Yaskawa INFORM job: OK_R2_O242(-90,180)OKKR.JBI

/JOB
//NAME OK_R2_O242(-90,180)OKKR
///FOLDERNAME X4
//POS
///NPOS 132,132,132,4,0,0
///TOOL 0
///POSTYPE PULSE
///PULSE
C00000=-1085,-105763,-105592,-1367,57789,79187
C00001=-48587,-61870,-56373,-37554,57186,71211
C00002=-109319,-98863,-81663,17130,36799,47258
C00003=-110499,-70978,-76585,14581,28064,55521
C00004=-114923,11399,-23396,32739,57115,42289
C00005=-116623,27529,-9023,35345,61036,36673
C00006=-106531,29443,-6029,23966,54360,54184
C00007=-107072,29107,-4870,24608,53702,53789
C00008=-107072,28853,-4001,24811,53095,53633
C00009=-107072,28916,-4224,24758,53250,53673
C00010=-107722,30543,-2610,25264,53294,53401
C00011=-107072,28916,-4224,24758,53250,53673
C00012=-111142,26244,-323,41203,47920,52388
C00013=-110370,28048,1439,40770,47447,52585
C00014=-111142,26244,-323,41203,47920,52388
C00015=-118906,20077,-8538,45056,52999,50729
C00016=-119909,26329,-1133,46362,52540,49898
C00017=-119909,26168,171,46853,51920,49532
C00018=-119909,26196,-79,46760,52037,49603
C00019=-119136,27214,914,46366,51584,49791
C00020=-119909,26334,-1167,46350,52555,49909
C00021=-114397,22245,-5862,42574,50447,51878
C00022=-114678,22860,-3308,43462,49647,51288
C00023=-115167,24031,-2185,43822,49818,51101
C00024=-114397,22245,-5862,42574,50447,51878
C00025=-121530,27687,-2626,46433,54487,50098
C00026=-123087,41300,13747,48930,53168,48397
C00027=-123087,41268,14126,49069,53001,48291
C00028=-123087,41187,15376,49530,52460,47945
C00029=-123087,41201,15124,49437,52567,48015
C00030=-122538,42735,16737,49268,52140,48077
C00031=-123087,41401,12757,48563,53611,48677
C00032=-122129,71626,35140,38253,65229,58469
C00033=-121790,71611,37598,38532,63876,58094
C00034=-121434,69636,35263,38247,64057,58328
C00035=-122129,71626,35140,38253,65229,58469
C00036=-120911,36076,-5205,37468,69020,59397
C00037=-115840,28901,-5746,41502,62039,42211
C00038=-98326,48101,7238,8655,64893,45952
C00039=-115260,32848,2305,42264,59563,41364
C00040=-114901,35009,3238,41874,59801,41652
C00041=-97533,41248,-17,1386,65111,50229
C00042=-97538,41207,-61,1389,65116,50227
C00043=-106518,42771,1588,20090,69082,39147
C00044=-114870,56219,16256,34532,77057,29376
C00045=-115508,58548,18881,34817,76955,29091
C00046=-119108,76539,39651,36547,75490,27151
C00047=-119068,69741,30113,36226,77407,27817
C00048=-119017,62946,18494,35839,80377,88071
C00049=-119017,62946,18494,34539,69439,88067
C00050=-120365,66463,30779,36511,65240,86054
C00051=-120262,68091,33866,36748,64342,85770
C00052=-120262,68091,33866,36748,64342,85770
C00053=-120199,73821,40919,37119,63187,85370
C00054=-119797,77336,44812,37019,63133,85550
C00055=-121282,70665,32992,36655,66863,86263
C00056=-119068,69741,30113,36226,77407,27817
C00057=-122206,59988,23685,43496,73319,20353
C00058=-127814,79238,36559,32495,95149,850
C00059=-120292,64376,19422,33176,77212,56642
C00060=-112530,30789,-557,20785,48585,51256
C00061=-109411,60829,14687,9556,77735,26746
C00062=-109666,62467,17842,9701,76678,26580
C00063=-109739,35424,4016,18642,47529,52303
C00064=-109346,36012,4533,18322,47429,52463
C00065=-111432,39361,576,18526,58483,53933
C00066=-120982,47505,9487,38936,66696,53604
C00067=-124164,44416,17003,51861,57678,49293
C00068=-125991,53710,27094,53356,57812,48240
C00069=-126351,53462,26814,53496,58041,48175
C00070=-128648,70270,46080,56033,57461,46239
C00071=-128914,63950,33868,51063,60408,47630
C00072=-125493,46290,11213,43702,62626,49802
C00073=-121024,34692,-8870,25769,64212,48636
C00074=-116968,-20453,-45092,25851,41430,48067
C00075=-118489,-78623,-76964,34127,32976,43558
C00076=-15896,-74508,-72271,-73191,84674,57421
C00077=-31461,-74136,-72097,-73237,111249,57325
C00078=-37199,-69408,-69826,-73614,107600,56062
C00079=3643,-76224,-106676,19950,71810,76872
C00080=-49550,-101636,-102264,-56737,88786,-31332
C00081=-138514,-74114,-82544,-4040,38797,-48213
C00082=-129498,7065,-37023,-9065,67369,-37181
C00083=-133542,65003,16374,-22570,90358,-433
C00084=-140622,86165,36573,-15496,97977,30873
C00085=-140802,90119,43938,-15362,95529,31124
C00086=-140802,89712,44636,-15338,94910,31202
C00087=-140802,89824,44435,-15345,95084,31180
C00088=-141302,92318,47595,-15241,94356,31104
C00089=-140802,90328,43607,-15371,95825,31086
C00090=-139449,100407,57298,-15497,92942,31904
C00091=-140520,104512,63149,-15296,91307,31746
C00092=-140782,103254,61503,-15262,91612,31621
C00093=-140520,104512,63149,-15296,91307,31746
C00094=-139554,101999,57136,-15503,93810,31760
C00095=-146528,71128,18474,-14629,100276,28663
C00096=-157576,61757,12077,-2365,89224,8186
C00097=-158570,72432,22020,-167,94145,8287
C00098=-158570,72037,22464,-167,93669,8287
C00099=-158570,72148,22336,-167,93805,8287
C00100=-157930,73423,23870,-319,93520,8487
C00101=-158570,72260,22211,-167,93940,8288
C00102=-159049,73117,23241,-53,93746,8137
C00103=-159487,76071,26810,51,93068,8000
C00104=-159049,73117,23241,-53,93746,8137
C00105=-152305,60889,6833,-1672,97624,10189
C00106=-140378,92804,43752,-12660,95661,26275
C00107=-136628,131083,97606,-23032,87536,68506
C00108=-138246,133972,103985,-22893,84834,68434
C00109=-138116,121410,87047,-22215,87119,66148
C00110=-138089,120831,86265,-22218,87298,66125
C00111=-139222,110925,72109,-17859,93005,38128
C00112=-141573,89787,44718,-13729,93335,28318
C00113=-147118,72338,23336,-11669,95813,24471
C00114=-147124,72286,23273,-11668,95824,24468
C00115=-156033,62541,11743,1459,94557,7242
C00116=-162183,69089,19251,9179,95274,-2750
C00117=-162693,76607,28216,6950,92750,113
C00118=-162306,74109,24034,6874,94001,304
C00119=-159278,70446,19892,6162,94440,1277
C00120=-158882,69844,19507,6067,94341,1397
C00121=-162546,67834,20044,10120,87741,415
C00122=-153853,64460,11220,-3191,96050,12949
C00123=-153394,69903,19674,-3303,93668,13156
C00124=-150617,75820,26688,-3977,92508,14059
C00125=-150141,75566,26453,-4094,92547,14205
C00126=-143887,90860,45319,-9758,90806,22100
C00127=-142426,78831,26541,-11541,97051,24087
C00128=-145972,26725,-27800,-4713,87219,24751
C00129=-154694,-16289,-62866,3052,73548,23707
C00130=-178421,-116488,-119781,18026,60210,14368
C00131=-104141,-125863,-97896,-54468,42310,-61417
BC00000=193639,675452,895426
BC00001=148805,682642,173588
BC00002=141606,703754,90547
BC00003=133760,726761,53
BC00004=133760,726761,53
BC00005=133760,726761,53
BC00006=133760,726761,53
BC00007=133760,726761,53
BC00008=133760,726761,53
BC00009=133760,726761,53
BC00010=133760,726761,53
BC00011=133760,726761,53
BC00012=133760,726761,53
BC00013=133760,726761,53
BC00014=133760,726761,53
BC00015=133760,726761,53
BC00016=133760,726761,53
BC00017=133760,726761,53
BC00018=133760,726761,53
BC00019=133760,726761,53
BC00020=133760,726761,53
BC00021=133760,726761,53
BC00022=133760,726761,53
BC00023=133760,726761,53
BC00024=133760,726761,53
BC00025=133760,726761,53
BC00026=133760,726761,53
BC00027=133760,726761,53
BC00028=133760,726761,53
BC00029=133760,726761,53
BC00030=133760,726761,53
BC00031=133760,726761,53
BC00032=133760,726761,53
BC00033=133760,726761,53
BC00034=133760,726761,53
BC00035=133760,726761,53
BC00036=133760,726761,53
BC00037=122204,725818,53
BC00038=122204,725818,53
BC00039=122204,725818,53
BC00040=122204,725818,53
BC00041=122204,725818,53
BC00042=122204,725818,53
BC00043=122204,725818,53
BC00044=122204,725818,53
BC00045=122204,725818,53
BC00046=122204,725818,53
BC00047=122204,725818,53
BC00048=122204,725818,53
BC00049=122204,725818,53
BC00050=122204,725818,53
BC00051=122204,725818,50
BC00052=122204,725818,50
BC00053=122204,725818,50
BC00054=122204,725818,50
BC00055=122204,725818,50
BC00056=122204,725818,53
BC00057=122204,725818,53
BC00058=171344,723534,1465
BC00059=151059,717900,51
BC00060=151059,717900,51
BC00061=151058,717899,53
BC00062=151058,717899,53
BC00063=151059,717900,51
BC00064=151059,717900,51
BC00065=151059,717900,51
BC00066=151059,717900,51
BC00067=151059,717900,51
BC00068=151059,717899,51
BC00069=151059,717900,51
BC00070=151059,717900,51
BC00071=151059,717900,51
BC00072=151059,717900,51
BC00073=150319,720693,10790
BC00074=145099,682085,7405
BC00075=145099,683773,7405
BC00076=139754,687631,3940
BC00077=139754,686805,3940
BC00078=139920,676862,3936
BC00079=199464,674570,1075173
BC00080=228966,680708,53
BC00081=305664,727709,53
BC00082=305664,727709,53
BC00083=337516,744483,53
BC00084=364852,758879,53
BC00085=364852,758879,53
BC00086=364852,758879,53
BC00087=364852,758879,53
BC00088=364852,758879,53
BC00089=364852,758879,53
BC00090=364852,758879,53
BC00091=364852,758879,53
BC00092=364852,758879,53
BC00093=364852,758879,53
BC00094=364852,758879,53
BC00095=364852,758879,53
BC00096=364852,758879,53
BC00097=364852,758879,53
BC00098=364852,758879,53
BC00099=364852,758879,53
BC00100=364852,758879,53
BC00101=364852,758879,53
BC00102=364852,758879,53
BC00103=364852,758879,53
BC00104=364852,758879,53
BC00105=364852,758879,53
BC00106=364852,758879,53
BC00107=364852,758879,53
BC00108=364852,758879,53
BC00109=364852,758879,53
BC00110=364852,758879,53
BC00111=364852,758879,53
BC00112=364852,758879,53
BC00113=364852,758879,53
BC00114=364852,758879,53
BC00115=364852,758879,53
BC00116=364852,758879,53
BC00117=364852,758879,53
BC00118=364852,758879,53
BC00119=364852,758879,53
BC00120=364852,758879,53
BC00121=364852,758879,53
BC00122=364852,758879,53
BC00123=364852,758878,49
BC00124=364852,758878,49
BC00125=364852,758878,49
BC00126=364852,758878,49
BC00127=364852,758878,49
BC00128=364852,758878,49
BC00129=364852,758878,49
BC00130=364852,758878,49
BC00131=299903,700532,95945
EC00000=-798141,218
EC00001=-798073,1230
EC00002=-798113,641
EC00003=-798156,0
EC00004=-798156,0
EC00005=-798156,0
EC00006=-798156,0
EC00007=-798156,0
EC00008=-798156,0
EC00009=-798156,0
EC00010=-798156,0
EC00011=-798156,0
EC00012=-798156,0
EC00013=-798156,0
EC00014=-798156,0
EC00015=-798156,0
EC00016=-798156,0
EC00017=-798156,0
EC00018=-798156,0
EC00019=-798156,0
EC00020=-798156,0
EC00021=-798156,0
EC00022=-798156,0
EC00023=-798156,0
EC00024=-798156,0
EC00025=-798156,0
EC00026=-798156,0
EC00027=-798156,0
EC00028=-798156,0
EC00029=-798156,0
EC00030=-798156,0
EC00031=-798156,0
EC00032=-798156,0
EC00033=-798156,0
EC00034=-798156,0
EC00035=-798156,0
EC00036=-798156,0
EC00037=-798156,0
EC00038=-798156,0
EC00039=-798156,0
EC00040=-798156,0
EC00041=-798156,0
EC00042=-798156,0
EC00043=-798156,0
EC00044=-798156,0
EC00045=-798156,0
EC00046=-798156,0
EC00047=-798156,0
EC00048=-798156,0
EC00049=-798156,0
EC00050=-798156,0
EC00051=-798155,-2
EC00052=-798155,-2
EC00053=-798155,-2
EC00054=-798155,-2
EC00055=-798155,-2
EC00056=-798156,0
EC00057=-798156,0
EC00058=-798156,0
EC00059=-798155,0
EC00060=-798155,0
EC00061=-798156,0
EC00062=-798156,0
EC00063=-798155,0
EC00064=-798155,0
EC00065=-798155,0
EC00066=-798155,0
EC00067=-798155,0
EC00068=-798155,0
EC00069=-798155,0
EC00070=-798155,0
EC00071=-798155,0
EC00072=-798155,0
EC00073=-798155,0
EC00074=-798155,0
EC00075=-798155,0
EC00076=-798155,0
EC00077=-878588,219672
EC00078=-886883,834249
EC00079=-798156,1112951
EC00080=-798156,1112951
EC00081=-798156,1112951
EC00082=-798156,1112951
EC00083=-798156,1112951
EC00084=-798156,1112951
EC00085=-798156,1112951
EC00086=-798156,1112951
EC00087=-798156,1112951
EC00088=-798156,1112951
EC00089=-798156,1112951
EC00090=-798156,1112951
EC00091=-798156,1112951
EC00092=-798156,1112951
EC00093=-798156,1112951
EC00094=-798156,1112951
EC00095=-798156,1112951
EC00096=-798156,1112951
EC00097=-798156,1112951
EC00098=-798156,1112951
EC00099=-798156,1112951
EC00100=-798156,1112951
EC00101=-798156,1112951
EC00102=-798156,1112951
EC00103=-798156,1112951
EC00104=-798156,1112951
EC00105=-798156,1112951
EC00106=-798156,1112951
EC00107=-798156,1112951
EC00108=-798156,1112951
EC00109=-798156,1112951
EC00110=-798156,1112951
EC00111=-798156,1112951
EC00112=-798156,1112951
EC00113=-798156,1112951
EC00114=-798156,1112951
EC00115=-798156,1112951
EC00116=-798156,1112951
EC00117=-798156,1112951
EC00118=-798156,1112951
EC00119=-798156,1112951
EC00120=-798156,1112951
EC00121=-798156,1112951
EC00122=-798156,1112951
EC00123=-798155,1112954
EC00124=-798155,1112954
EC00125=-798155,1112954
EC00126=-798155,1112954
EC00127=-798155,1112954
EC00128=-798155,1112954
EC00129=-798155,1112954
EC00130=-798155,1112954
EC00131=-798156,1112951
///POSTYPE BASE
///RECTAN
///RCONF 0,0,0,0,0,0,0,0,0,0,0,0,0,0,0,0,0,0,0,0,0,0,0,0
P00006=0.222,-3.123,-1.508,0.0000,0.0000,0.0000
P00021=-0.225,-6.128,-0.405,0.0000,0.0000,0.0000
P00022=0.222,-3.123,-1.508,0.0000,0.0000,0.0000
P00023=0.143,-0.036,0.682,0.0000,0.0000,0.0000
//INST
///DATE 2024/11/06 09:54
///ATTR SC,RW
///GROUP1 RB1,BS1
///GROUP2 ST1
NOP
'OK_r2_O24.2(-90,180)
'-90,0
MOVJ C00000 BC00000 VJ=100.00  +MOVJ EC00000 VJ=100.00
MOVJ C00001 BC00001 VJ=100.00  +MOVJ EC00001 VJ=25.00
MOVJ C00002 BC00002 VJ=100.00  +MOVJ EC00002 VJ=25.00
MOVJ C00003 BC00003 VJ=100.00  +MOVJ EC00003 VJ=100.00
MOVJ C00004 BC00004 VJ=100.00  +MOVJ EC00004 VJ=25.00
'Path S1574
SFTOF3D
MOVJ C00005 BC00005 VJ=100.00  +MOVJ EC00005 VJ=100.00
MOVL C00006 BC00006 V=166.7  +MOVJ EC00006 VJ=100.00
SMOVL C00007 BC00007 V=100.0  +MOVJ EC00007
SREFP 3 C00008 BC00008  +REFP EC00008
CALL JOB:SEARCH-R1-S13D
SET P021 P006
SFTON3D P021
SMOVL C00009 BC00009 V=100.0  +MOVJ EC00009
SREFP 3 C00010 BC00010  +REFP EC00010
CALL JOB:SEARCH-R1-S13D
SET P021 P006
SFTON3D P021
SMOVL C00011 BC00011 V=100.0  +MOVJ EC00011
SMOVL C00012 BC00012 V=200.0  +MOVJ EC00012
SREFP 3 C00013 BC00013  +REFP EC00013
CALL JOB:SEARCH-R1-S13D
SET P021 P006
SFTON3D P021
SMOVL C00014 BC00014 V=100.0  +MOVJ EC00014
SFTOF3D
MOVL C00015 BC00015 V=400.0  +MOVJ EC00015 VJ=100.00
SMOVL C00016 BC00016 V=133.3  +MOVJ EC00016
SREFP 3 C00017 BC00017  +REFP EC00017
CALL JOB:SEARCH-R1-S13D
SET P022 P006
SFTON3D P022
SMOVL C00018 BC00018 V=100.0  +MOVJ EC00018
SREFP 3 C00019 BC00019  +REFP EC00019
CALL JOB:SEARCH-R1-S13D
SET P022 P006
SFTON3D P022
SMOVL C00020 BC00020 V=100.0  +MOVJ EC00020
SMOVL C00021 BC00021 V=200.0  +MOVJ EC00021
SMOVL C00022 BC00022 V=133.3  +MOVJ EC00022
SREFP 3 C00023 BC00023  +REFP EC00023
CALL JOB:SEARCH-R1-S13D
SET P022 P006
SFTON3D P022
SMOVL C00024 BC00024 V=100.0  +MOVJ EC00024
SFTOF3D
SMOVL C00025 BC00025 V=333.3  +MOVJ EC00025
SMOVL C00026 BC00026 V=166.7  +MOVJ EC00026
SMOVL C00027 BC00027 V=100.0  +MOVJ EC00027
SREFP 3 C00028 BC00028  +REFP EC00028
CALL JOB:SEARCH-R1-S13D
SET P023 P006
SFTON3D P023
SMOVL C00029 BC00029 V=100.0  +MOVJ EC00029
SREFP 3 C00030 BC00030  +REFP EC00030
CALL JOB:SEARCH-R1-S13D
SET P023 P006
SFTON3D P023
SMOVL C00031 BC00031 V=100.0  +MOVJ EC00031
SMOVL C00032 BC00032 V=200.0  +MOVJ EC00032
SMOVL C00033 BC00033 V=166.7  +MOVJ EC00033
SREFP 3 C00034 BC00034  +REFP EC00034
CALL JOB:SEARCH-R1-S13D
SET P023 P006
SFTON3D P023
SMOVL C00035 BC00035 V=200.0  +MOVJ EC00035
SFTOF3D
SMOVL C00036 BC00036 V=500.0  +MOVJ EC00036
'Path W1575
SFTOF3D
SFTON3D P021
MOVJ C00037 BC00037 VJ=100.00  +MOVJ EC00037 VJ=100.00
SMOVL C00038 BC00038 V=166.7 PL=0  +MOVJ EC00038
SREFP 1 C00039 BC00039  +REFP EC00039
SREFP 2 C00040 BC00040  +REFP EC00040
MACRO1 MJ#(0) ARGF9
ARCON
SMOVL C00041 BC00041 V=10.0  +MOVJ EC00041
SMOVC C00042 BC00042 V=10.0  +MOVJ EC00042
SMOVC C00043 BC00043 V=10.0  +MOVJ EC00043
SFTON3D P022
SMOVC C00044 BC00044 V=10.0  +MOVJ EC00044
SMOVC C00045 BC00045 V=10.0  +MOVJ EC00045
SFTON3D P023
SMOVL C00046 BC00046 V=10.0  +MOVJ EC00046
ARCOF
SMOVL C00047 BC00047 V=400.0  +MOVJ EC00047
SMOVL C00048 BC00048 V=400.0  +MOVJ EC00048
SMOVL C00049 BC00049 V=400.0  +MOVJ EC00049
SMOVL C00050 BC00050 V=400.0  +MOVJ EC00050
SMOVL C00051 BC00051 V=166.7 PL=0  +MOVJ EC00051
ARCON
SMOVC C00052 BC00052 V=10.0  +MOVJ EC00052
SMOVC C00053 BC00053 V=10.0  +MOVJ EC00053
SMOVC C00054 BC00054 V=10.0  +MOVJ EC00054
ARCOF
SMOVL C00055 BC00055 V=333.3  +MOVJ EC00055
SMOVL C00056 BC00056 V=400.0  +MOVJ EC00056
SMOVL C00057 BC00057 V=1000.0  +MOVJ EC00057
SFTOF3D
'Path W1576
SFTOF3D
SFTON3D P021
SMOVL C00058 BC00058 V=133.3  +MOVJ EC00058
SFTOF3D
SFTON3D P021
SMOVL C00059 BC00059 V=133.3  +MOVJ EC00059
SMOVL C00060 BC00060 V=133.3 PL=0  +MOVJ EC00060
SREFP 1 C00061 BC00061  +REFP EC00061
SREFP 2 C00062 BC00062  +REFP EC00062
MACRO1 MJ#(0) ARGF9
ARCON
SMOVL C00063 BC00063 V=7.5  +MOVJ EC00063
SMOVL C00064 BC00064 V=7.5  +MOVJ EC00064
ARCOF
MOVL C00065 BC00065 V=166.7  +MOVJ EC00065 VJ=25.00
SFTOF3D
MOVL C00066 BC00066 V=250.0  +MOVJ EC00066 VJ=25.00
SFTON3D P022
SMOVL C00067 BC00067 V=133.3  +MOVJ EC00067
ARCON
SMOVL C00068 BC00068 V=7.5  +MOVJ EC00068
SMOVL C00069 BC00069 V=7.5  +MOVJ EC00069
ARCON
SFTON3D P023
SMOVL C00070 BC00070 V=7.5  +MOVJ EC00070
ARCOF
SMOVL C00071 BC00071 V=166.7  +MOVJ EC00071
SMOVL C00072 BC00072 V=400.0  +MOVJ EC00072
SFTOF3D
MOVJ C00073 BC00073 VJ=100.00  +MOVJ EC00073 VJ=100.00
MOVJ C00074 BC00074 VJ=100.00  +MOVJ EC00074 VJ=25.00
MOVJ C00075 BC00075 VJ=100.00  +MOVJ EC00075 VJ=25.00
MOVJ C00076 BC00076 VJ=100.00  +MOVJ EC00076 VJ=100.00
'-90,180
MOVJ C00077 BC00077 VJ=100.00  +MOVJ EC00077 VJ=100.00
MOVJ C00078 BC00078 VJ=100.00  +MOVJ EC00078 VJ=100.00
MOVJ C00079 BC00079 VJ=100.00  +MOVJ EC00079 VJ=100.00
CALL JOB:CLEAN-R1_KM_NEW
MOVJ C00080 BC00080 VJ=100.00  +MOVJ EC00080 VJ=25.00
MOVJ C00081 BC00081 VJ=100.00  +MOVJ EC00081 VJ=100.00
MOVJ C00082 BC00082 VJ=100.00  +MOVJ EC00082 VJ=25.00
'Path S1580
SFTOF3D
MOVJ C00083 BC00083 VJ=100.00  +MOVJ EC00083 VJ=100.00
MOVJ C00084 BC00084 VJ=100.00  +MOVJ EC00084 VJ=100.00
SMOVL C00085 BC00085 V=133.3  +MOVJ EC00085
SREFP 3 C00086 BC00086  +REFP EC00086
CALL JOB:SEARCH-R1-S13D
SET P021 P006
SFTON3D P021
SMOVL C00087 BC00087 V=100.0  +MOVJ EC00087
SREFP 3 C00088 BC00088  +REFP EC00088
CALL JOB:SEARCH-R1-S13D
SET P021 P006
SFTON3D P021
SMOVL C00089 BC00089 V=100.0  +MOVJ EC00089
SMOVL C00090 BC00090 V=166.7  +MOVJ EC00090
SMOVL C00091 BC00091 V=100.0  +MOVJ EC00091
SREFP 3 C00092 BC00092  +REFP EC00092
CALL JOB:SEARCH-R1-S13D
SET P021 P006
SFTON3D P021
SMOVL C00093 BC00093 V=100.0  +MOVJ EC00093
SMOVL C00094 BC00094 V=333.3  +MOVJ EC00094
SFTOF3D
SMOVL C00095 BC00095 V=333.3  +MOVJ EC00095
SMOVL C00096 BC00096 V=333.3  +MOVJ EC00096
SMOVL C00097 BC00097 V=100.0  +MOVJ EC00097
SREFP 3 C00098 BC00098  +REFP EC00098
CALL JOB:SEARCH-R1-S13D
SET P022 P006
SFTON3D P022
SMOVL C00099 BC00099 V=100.0  +MOVJ EC00099
SREFP 3 C00100 BC00100  +REFP EC00100
CALL JOB:SEARCH-R1-S13D
SET P022 P006
SFTON3D P022
SMOVL C00101 BC00101 V=100.0  +MOVJ EC00101
SMOVL C00102 BC00102 V=166.7  +MOVJ EC00102
SREFP 3 C00103 BC00103  +REFP EC00103
CALL JOB:SEARCH-R1-S13D
SET P022 P006
SFTON3D P022
SMOVL C00104 BC00104 V=100.0  +MOVJ EC00104
SFTOF3D
SMOVL C00105 BC00105 V=333.3  +MOVJ EC00105
MOVJ C00106 BC00106 VJ=100.00  +MOVJ EC00106 VJ=100.00
MOVJ C00107 BC00107 VJ=100.00  +MOVJ EC00107 VJ=100.00
MACRO1 MJ#(0) ARGF9
SFTON3D P021
SMOVL C00108 BC00108 V=133.3  +MOVJ EC00108
ARCON
SMOVL C00109 BC00109 V=10.0  +MOVJ EC00109
SMOVC C00110 BC00110 V=10.0  +MOVJ EC00110
SMOVC C00111 BC00111 V=10.0  +MOVJ EC00111
SMOVC C00112 BC00112 V=10.0  +MOVJ EC00112
SMOVL C00113 BC00113 V=10.0  +MOVJ EC00113
SMOVC C00114 BC00114 V=10.0  +MOVJ EC00114
SFTON3D P022
SMOVC C00115 BC00115 V=10.0  +MOVJ EC00115
SMOVC C00116 BC00116 V=10.0  +MOVJ EC00116
SMOVL C00117 BC00117 V=10.0  +MOVJ EC00117
ARCOF
SMOVL C00118 BC00118 V=166.7  +MOVJ EC00118
SFTOF3D
SMOVL C00119 BC00119 V=166.7  +MOVJ EC00119
SFTON3D P022
SMOVL C00120 BC00120 V=166.7  +MOVJ EC00120
ARCON
SMOVL C00121 BC00121 V=8.3  +MOVJ EC00121
ARCOF
SFTOF3D
SMOVL C00122 BC00122 V=166.7  +MOVJ EC00122
SFTON3D P021
SMOVL C00123 BC00123 V=10.0  +MOVJ EC00123
ARCON
SMOVL C00124 BC00124 V=8.3  +MOVJ EC00124
SMOVL C00125 BC00125 V=8.3  +MOVJ EC00125
SMOVL C00126 BC00126 V=8.3  +MOVJ EC00126
ARCOF
SMOVL C00127 BC00127 V=333.3  +MOVJ EC00127
SFTOF3D
MOVJ C00128 BC00128 VJ=100.00  +MOVJ EC00128 VJ=100.00
MOVJ C00129 BC00129 VJ=100.00  +MOVJ EC00129 VJ=100.00
MOVJ C00130 BC00130 VJ=100.00  +MOVJ EC00130 VJ=100.00
SFTOF3D
MOVJ C00131 BC00131 VJ=100.00  +MOVJ EC00131 VJ=100.00
END
